FUNCTION_BLOCK Test_TStreamAdd_Read_REAL_CheckAlignment EXTENDS T_UnitTestBase
VAR
    Stream  : T_Stream(StreamLength := 2);
    ArgType : E_ArgTypeId := E_ArgTypeId.Type_REAL;
END_VAR

{attribute 'analysis' := '-33'} // inhibit unused variable warning
METHOD RunTest
IF Retest THEN
    SUPER^.Init();
END_IF

IF TestCompleted THEN
    RETURN;
END_IF

F_Inc(CycleCount);
IF CycleCount > 1000 THEN
    Fail(Message := 'Timeout');
END_IF

Stream.Init(2);

Stream.Add_BYTE(123);// add a byte to test alignment checks...
Stream.Add_REAL(1.234567);

Stream.SetReadPosition(0);

Stream.Read_BYTE();

// check next value...	
AssertEquals_REAL(Expected     := 1.234567,
                            Actual       := Stream.Read_REAL(),
                            Delta        := 0.000001,
                            Message := 'Stream.Read_REAL()');

// check we are at the end of the stream..							
AssertEquals_UDINT(Expected     := Stream.StreamLength,
                             Actual       := Stream.ReadPosition,
                             Message := 'Stream.ReadPosition');

TestCompleted := TRUE;
END_METHOD

END_FUNCTION_BLOCK

(* stored: Version 1.1.0.1, ProductVersion 3.1.4024.15
   POU Test_TStreamAdd_Read_REAL_CheckAlignment: Id {2b7e2bb1-1fbc-4e1f-a942-1bad658be938}, SpecialFunc None
   Method RunTest: Id {e430165a-f041-4a2c-87fa-cff11ef2f96e} *)
